// TIA Portal V18 export
// export: Created 2025-12-01T17:50:33.4250553Z, ExportSetting None, DisplayName Totally Integrated Automation Portal, DisplayVersion V18 Update 5, DisplayName TIA Portal Openness, DisplayVersion V18 Update 5, DisplayName TIA Portal Teamcenter Gateway, DisplayVersion V18, DisplayName TIA Portal Version Control Interface, DisplayVersion V18, DisplayName STEP 7 Professional, DisplayVersion V18 Update 5, DisplayName STEP 7 Safety, DisplayVersion V18, DisplayName WinCC Professional, DisplayVersion V18 Update 5
DATA_BLOCK "ST10_GlobalError"   // DB1066
{ S7_Optimized_Access := 'FALSE' }
// stored: AutoNumber false
   VAR RETAIN
      COM : Struct
         MainPneumaticPressure1NOK : Bool;   // Main Pneumatic pressure 1 NOK,pls check inptut Ix.x,then check if the main valve is opened
         MainPneumaticPressure2NOK : Bool;   // Main Pneumatic pressure 2 NOK,pls check inptut Ix.x,then check if the main valve is opened
         MainPneumaticPressure3NOK : Bool;   // Main Pneumatic pressure 3 NOK,pls check inptut Ix.x,then check if the main valve is opened
         StationNotInHP : Bool;   // Station not in Home position,can't start cycle,pls check the Home positiong state
         CabinetTemperatureNotOk : Bool;   // Cabinet Temperature not OK, please check input Ix.x,then check if the cooling and fan is working
         CoolingUnitNotOk : Bool;   // Cooling unit not OK,pls check input Ix.x,then check if the cooling and fan is working
         RotateTablePositionNOK : Bool;   // The position of the rotate table is not correct after change mode.pls reset position by manual
         RotateTableNotInPosition : Bool;   // No position signal after rotate table Stopped,please check table position and input Ix.x
         StationHardwareError : Bool;
         ChangeStyleError : Bool;
         Reserve3 : Bool;
         Reserve4 : Bool;
         Reserve5 : Bool;
         Reserve6 : Bool;
         Reserve7 : Bool;
         Reserve8 : Bool;
         Reserve : Array[1..4, 0..15] of Bool;
      END_STRUCT;
      Hardware : Struct
         PNSlaveStation01 : Array[1..10] of Struct
            Error : Bool;   // PLC Local Module Error,please check the error module,PLC hardware configuration and online monitor the PLC error message
            Reserve1 : Bool;
            Reserve2 : Bool;
         END_STRUCT;
         COMM : Array[1..5] of Struct   // Communication
            CommunicationError : Bool;   // Serial Communication error,please check power, hardware configuration and connection cable
            NoReceive : Bool;   // Serial Communication receive no information, please check the module settings and communication equipment is the same, check the communication line is the intersection or straight line
            ReceiveWrong : Bool;   // Serial Communication receive the information is wrong, please check the data area is updated in real time
            Reserve1 : Bool;
            Reserve2 : Bool;
         END_STRUCT;
         PNSlaveStation02 : Array[1..10] of Struct   // Substation
            Error : Bool;   // SubStation Missing, please check power, hardware configuration and connection cable
            Reserve1 : Bool;   // SubStation error, please check Slave error code, check the error information in the PLC online hardware
            Reserve2 : Bool;
            Reserve3 : Bool;
         END_STRUCT;
         PNSlaveStation03 : Array[1..10] of Struct   // Remote I/O Error (远程I/O错误）
            Error : Bool;   // Remote I/O communication error, please check the power and communication cable, check the hardware configuration of PLC
            Reserve1 : Bool;   // Remote I/O error, please online monitor the PLC error message
            Reserve2 : Bool;
            Reserve3 : Bool;
         END_STRUCT;
         ValveIsland : Array[1..5] of Struct   // Valve Island Error（阀岛错误）
            SystemError : Bool;   // Valve island error, pls check the error code , check the error information in the PLC online hardware
            OffLine : Bool;   // Valve island is lost, pls check the island's cable , check valve island in PLC configuration and the actual agreement
            Reserve1 : Bool;
            Reserve2 : Bool;
         END_STRUCT;
      END_STRUCT;
      Safety : Struct
         "Robot 1 Estop" : Bool;   // Safety circuit not OK,pls check input Ix.x,then check if the safety circuit control on
         "Robot 2 Estop" : Bool;   // E-stop safety circuit not OK, please check input Ix.x, then reset safety circurt
         HMIEstopPBActivated : Bool;   // HMI Estop PB Activated，pls check input Ix.x,then check Estop button,if Estop button is close,pls open the Estop button
         TableEstopPB1Activated : Bool;   // HTable Estop PB1 Activated，pls check input Ix.x,then check Estop button,if Estop button is close,pls open the Estop button
         TableEstopPB2Activated : Bool;   // Table Estop PB2 Activated，pls check input Ix.x,then check Estop button,if Estop button is close,pls open the Estop button
         TableEstopPB3Activated : Bool;   // Table Estop PB3 Activated，pls check input Ix.x,then check Estop button,if Estop button is close,pls open the Estop button
         TableEstopPB4Activated : Bool;   // Table Estop PB4 Activated，pls check input Ix.x,then check Estop button,if Estop button is close,pls open the Estop button
         TableEstopPB5Activated : Bool;   // Table Estop PB5 Activated，pls check input Ix.x,then check Estop button,if Estop button is close,pls open the Estop button
         TableEstopPB6Activated : Bool;   // Table Estop PB6 Activated，pls check input Ix.x,then check Estop button,if Estop button is close,pls open the Estop button
         EStopSafety : Bool;
         TableEstopPB7Activated : Bool;
         TableEstopPB8Activated : Bool;
         TableEstopPB9Activated : Bool;
         StoveEstopActivated : Bool;
         "Robot 3 Estop" : Bool;
         Reserve9 : Bool;
         Reserve : Array[1..4, 0..15] of Bool;
      END_STRUCT;
      SafetyDoor : Struct
         "Type" : Array[1..5] of Struct   // Safety Door circuit type
            NotOk : Bool;   // Safety Door type [*] circuit not OK, please check input Ix.x, then reset safety circurt
            OpenInRunning : Bool;   // The safety door is opened when device Running,pls power on than initialize device
            Reserve1 : Bool;
            Reserve2 : Bool;
         END_STRUCT;
         No : Array[1..9] of Struct   // SafetyDoorNumber
            NotLock : Bool;   // Safety door lock is not lock，pls check input Ix.x，then check safety door lock output Qx.x
            Notlocked : Bool;   // Safety door lock is not unlock，pls check input Ix.x，then check safety door lock output Qx.x
            NotClose : Bool;   // Safety door is not close,pls check satety door lock position
            Reserve1 : Bool;
            Reserve2 : Bool;
         END_STRUCT;
         MaterialDoor : Struct
            NotLock_1 : Bool;
            NotClose_1 : Bool;
            NotLock_2 : Bool;
            NotClose_2 : Bool;
            NotLock_3 : Bool;
            NotClose_3 : Bool;
            NotLock_4 : Bool;
            NotClose_4 : Bool;
            NotLock_5 : Bool;
            NotClose_5 : Bool;
            NotLock_6 : Bool;
            NotClose_6 : Bool;
            NotLock_7 : Bool;
            NotClose_7 : Bool;
            NotLock_8 : Bool;
            NotClose_8 : Bool;
         END_STRUCT;
      END_STRUCT;
      LightCurtain : Array[1..5] of Struct
         ActivatedInRunning : Bool;   // Light curtain is Activated when device Running, pls power on than initialize device
         ActivatedInRotTableRun : Bool;   // Light curtain is Activated when rotate table running,please press the reset button to rotate the rotate table to position
         Error : Bool;   // Light curtain error,pls check the light curtain connection or check the error code
         Reserve1 : Bool;
         Reserve2 : Bool;
      END_STRUCT;
      Product : Array[1..5] of Struct
         TypeSelectionError : Bool;   // Product Type selection error,pls select the proper type
         TypeWrong : Bool;   // Product is not match current model, please make sure the product model is entered correctly
         NotforStation : Bool;   // Product not for this station,pls check if the Product is proper
         TypeAutoChangeError : Bool;
         Reserve2 : Bool;
      END_STRUCT;
      Fixture : Array[1..10] of Struct
         PositionError : Bool;   // Fixture [*] position error,pls put the fixture on proper positon
         TypeError : Bool;   // Fixture [*] tpye error,pls put the correct fixture into the tooling
         Reserve1 : Bool;
         Reserve2 : Bool;
      END_STRUCT;
      Breaker : Struct   // Power Breaker
         Trip : Array[1..16] of Bool;   // Breaker tripped, please check input Ix.x
      END_STRUCT;
   END_VAR
BEGIN
END_DATA_BLOCK
